# EPICS StreamDevice protocol: data/devcybaman.proto
InTerminator = ACK;
OutTerminator = CR;

initialize {
    out "A";
    in "";
}

getA {
	out "M101";
	in "%f";
}

getB {
	out "M201";
	in "%f";
}

getC {
	out "M301";
	in "%f";
}
